FUNCTION_BLOCK XtsDisableSequence IMPLEMENTS ITask
VAR_INPUT
END_VAR
VAR_OUTPUT
END_VAR
VAR
	_collisionGroup : ICollisionGroup;
	removeAllAxes : RemoveAllMoverFromGroup(_collisionGroup);
	grpStop : StopMoverGroup(_collisionGroup);
	State : INT;
	DisableTrigger: BOOL;
	moverNumbers : DINT := 1;
	AllMoversDisabled: BOOL;
	_busy : BOOL;
	_done : BOOL;
	_Error : BOOL;
	
	Logger : TcMessage_Ext;
END_VAR
VAR_IN_OUT
	arrMovers : ARRAY[*] OF IMover;
END_VAR

CASE State OF
	0:
		IF DisableTrigger THEN
			DisableTrigger := FALSE;
			_busy := TRUE;
			_done := FALSE;
			_Error := FALSE;
			IF _collisionGroup.GroupState = CAGroupStatus.mcGroupStateMoving THEN
				Logger.Send(TC_EVENTS.XtsCAGroupEvents.CAGroupStop,'');
				grpStop.Execute();
				State := 10;
			ELSE
				State := 20;
				removeAllAxes.RemoveAllMover();
				Logger.Send(TC_EVENTS.XtsCAGroupEvents.CaGroupRemoveMovers,'');
			END_IF
		END_IF
		
	10:
		IF grpStop.Done THEN
			State := 20;
			Logger.Send(TC_EVENTS.XtsCAGroupEvents.CaGroupRemoveMovers,'');
			removeAllAxes.RemoveAllMover();
		END_IF
	
	20:
		IF removeAllAxes.Done THEN
			FOR moverNumbers := LOWER_BOUND(arrMovers,1) TO UPPER_BOUND(arrMovers,1) DO
				arrMovers[moverNumbers].IdentInGroup := 0;
				arrMovers[moverNumbers].DisableAxis();
			END_FOR
			State := 30;
		END_IF
		
	30:
		AllMoversDisabled := TRUE;
		FOR moverNumbers := LOWER_BOUND(arrMovers,1) TO UPPER_BOUND(arrMovers,1) DO
			AllMoversDisabled := TRUE AND NOT arrMovers[moverNumbers].isEnabled();
		END_FOR
		IF AllMoversDisabled THEN
			logger.Send(TC_EVENTS.XtsCAGroupEvents.AllMoversDisabled,'');
			State := 40;
			_collisionGroup.Disable();
			logger.Send(TC_EVENTS.XtsCAGroupEvents.CAGroupDisable,'');
		END_IF
	40:
		IF _collisionGroup.GroupState = CAGroupStatus.mcGroupStateErrorStop THEN
			_collisionGroup.Reset();
			Logger.Send(TC_EVENTS.XtsCAGroupEvents.CAGroupReset,'');
		END_IF	
		State := 50;
		
	50:
		IF _collisionGroup.GroupState = 1 THEN
			State := 0;
			grpStop.Deceleration := Tc3_Mc3Definitions.MC_DEFAULT;
			grpStop.Jerk := Tc3_Mc3Definitions.MC_DEFAULT;
			
			_busy := FALSE;
			_done := true;
		END_IF
END_CASE

removeAllAxes();
grpStop();

METHOD Abort : BOOL
DisableTrigger := FALSE;
State := 0;
removeAllAxes.Abort();
grpStop.Abort();
END_METHOD

PROPERTY Busy : BOOL
GET
Busy := _busy;
END_GET
END_PROPERTY

METHOD Disable : BOOL
VAR_INPUT
END_VAR
DisableTrigger := true;
END_METHOD

PROPERTY Done : BOOL
GET
Done := _done;
END_GET
END_PROPERTY

PROPERTY Error : BOOL
GET
Error := _Error;
END_GET
END_PROPERTY

METHOD FB_init : BOOL
VAR_INPUT
	bInitRetains : BOOL; // if TRUE, the retain variables are initialized (warm start / cold start)
	bInCopyCode : BOOL;  // if TRUE, the instance afterwards gets moved into the copy code (online change)
	collisionGroup : ICollisionGroup;
END_VAR
_collisionGroup := collisionGroup;
removeAllAxes.FB_init(FALSE, FALSE, CAGroup := collisionGroup);
grpStop.FB_init(FALSE,FALSE,CAGroup := collisionGroup);
END_METHOD

METHOD SetEmergencyDynamics : BOOL
VAR_INPUT
END_VAR
grpStop.Deceleration := Tc3_Mc3Definitions.MC_MAXIMUM;
grpStop.Jerk := Tc3_Mc3Definitions.MC_MAXIMUM;
END_METHOD

END_FUNCTION_BLOCK

(* stored: Version 1.1.0.1, ProductVersion 3.1.4024.12
   POU XtsDisableSequence: Id {73e2f204-8f47-4c35-9b5f-a5e50b2f6f82}, SpecialFunc None
   Method Abort: Id {afd537cd-f397-4f71-a0b8-6dd2d52942e4}
   Property Busy: Id {fc07d329-127f-40be-b9dd-9f15379f97c1}
   Get Get: Id {9dd46cfd-26e2-4b1d-9cfd-59dc125dbe84}
   Method Disable: Id {d8277baf-d0a5-4ca3-b9d2-183e530222af}
   Property Done: Id {efc20aa9-c110-4223-9726-36ce2db4f287}
   Get Get: Id {c2112fc9-a6f8-4cc4-b638-2d26ce808170}
   Property Error: Id {19dd2892-ce5c-4277-bdea-9eefed81895d}
   Get Get: Id {286361e3-d2d3-4160-b40e-98196d8fec86}
   Method FB_init: Id {2df29c4c-50b6-4b7a-96ef-c07bbbce5982}
   Method SetEmergencyDynamics: Id {62e6980a-ad39-4f6d-bfa3-13e514d9c054} *)
